RESOURCE RES0 : EMB_RES_ECO
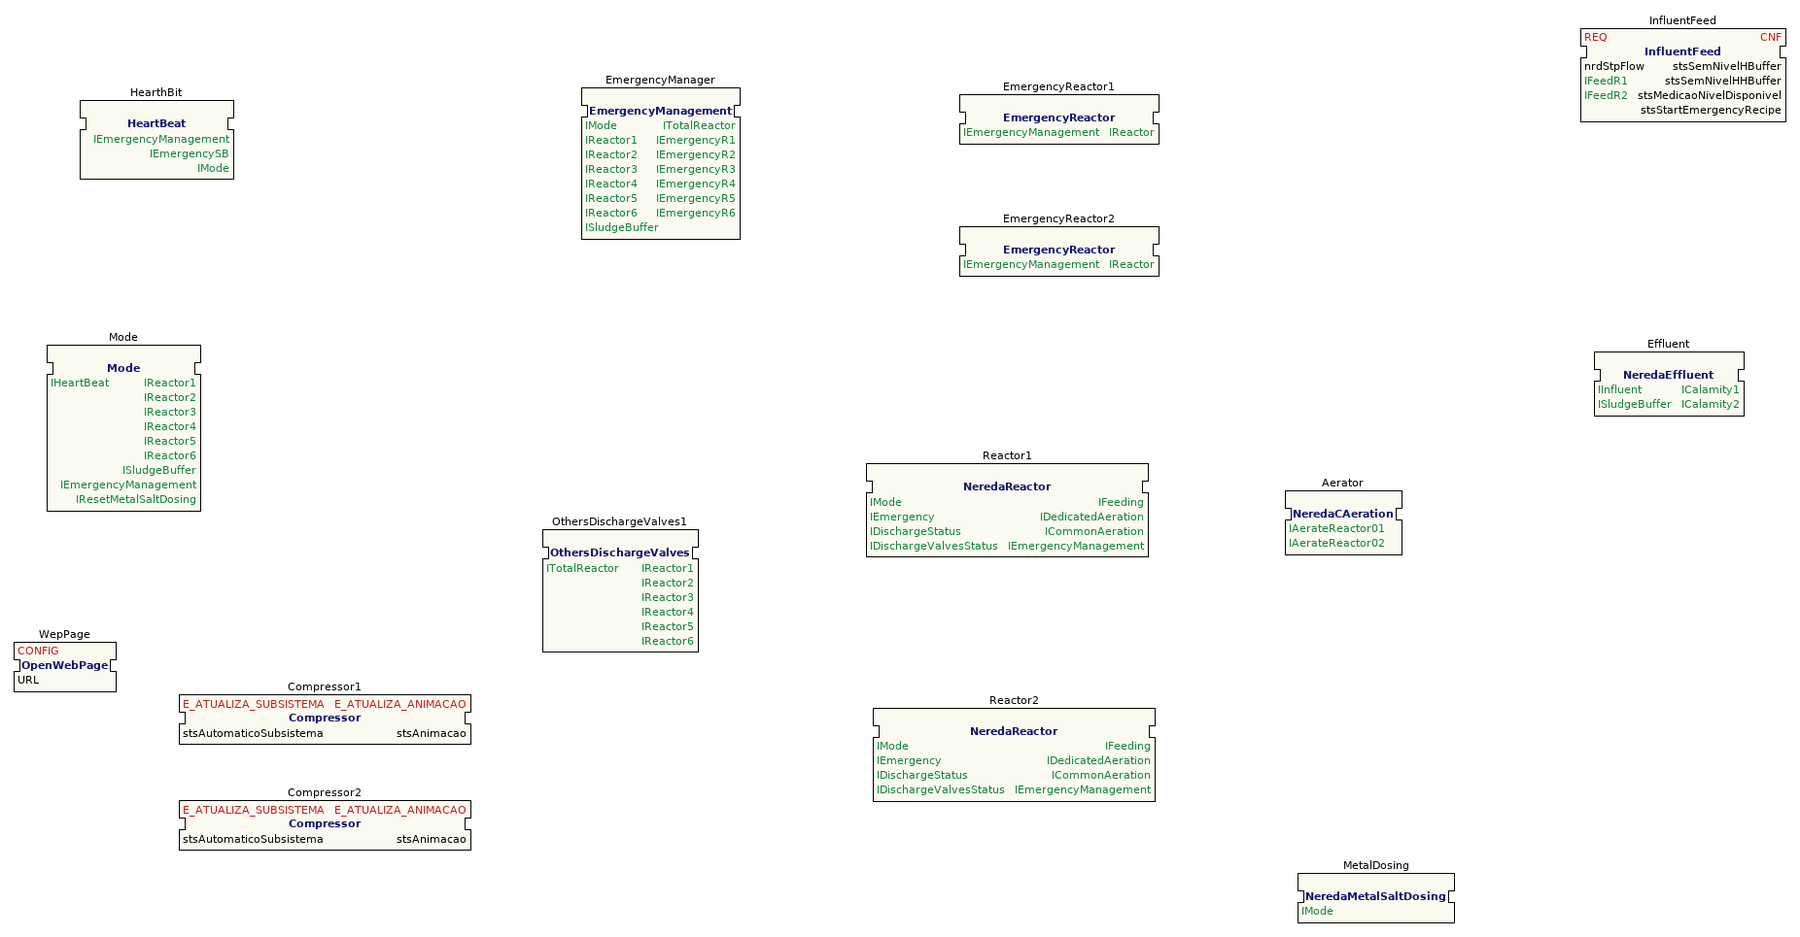
  FBS
    Reactor1 : NeredaReactor;
    Reactor2 : NeredaReactor;
    MetalDosing : NeredaMetalSaltDosing;
    InfluentFeed : InfluentFeed;
    EmergencyManager : EmergencyManagement;
    EmergencyReactor1 : EmergencyReactor;
    EmergencyReactor2 : EmergencyReactor;
    Effluent : NeredaEffluent;
    Compressor1 : Compressor;
    Compressor2 : Compressor;
    Aerator : NeredaCAeration;
    Mode : Mode;
    WepPage : OpenWebPage;
    HearthBit : HeartBeat;
    OthersDischargeValves1 : OthersDischargeValves;
  END_FBS
END_RESOURCE
